PROGRAM MAIN
VAR
END_VAR

IF OPC.bBit OR OPC.sMetin = 'Başla' THEN
	OPC.nSayi	:= OPc.nSayi + 1;
END_IF

END_PROGRAM

(* stored: Version 1.1.0.1, ProductVersion 3.1.4024.6
   POU MAIN: Id {ad288373-e3bd-45f4-9f90-28bbc0bfc537}, SpecialFunc None *)
